FUNCTION_BLOCK ButtonsPanel (* Composite Function Block Type *)
  (* Standard: 61499-2 *)
  (* Version 0.0, 7/13/2016, Andrei, nxtControl GmbH, template *)
  PACKAGE Main;
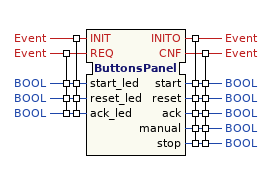
  EVENT_INPUT
    INIT WITH start_led, reset_led, ack_led; (* Initialization Request *)
    REQ WITH start_led, reset_led, ack_led; (* Normal Execution Request *)
  END_EVENT
  EVENT_OUTPUT
    INITO WITH start, reset, ack, manual, stop; (* Initialization Confirm *)
    CNF WITH start, reset, ack, manual, stop; (* Execution Confirmation *)
  END_EVENT
  VAR_INPUT
    start_led : BOOL; (* Input event qualifier *)
    reset_led : BOOL;
    ack_led : BOOL;
  END_VAR
  VAR_OUTPUT
    start : BOOL; (* Output event qualifier *)
    reset : BOOL;
    ack : BOOL;
    manual : BOOL;
    stop : BOOL;
  END_VAR
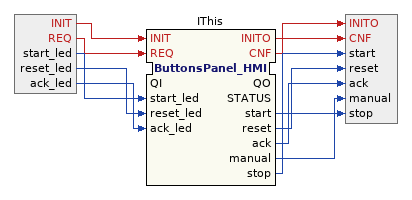
  FBS
    IThis : ButtonsPanel_HMI;
  END_FBS
  EVENT_CONNECTIONS
    INIT TO IThis.INIT;
    REQ TO IThis.REQ;
    IThis.INITO TO INITO;
    IThis.CNF TO CNF;
  END_CONNECTIONS
  DATA_CONNECTIONS
    start_led TO IThis.start_led;
    reset_led TO IThis.reset_led;
    ack_led TO IThis.ack_led;
    IThis.start TO start;
    IThis.reset TO reset;
    IThis.ack TO ack;
    IThis.manual TO manual;
    IThis.stop TO stop;
  END_CONNECTIONS
END_FUNCTION_BLOCK
